TYPE ST_IPCDiagParamSpec :
STRUCT
	eParam: E_IPCDiag_ParameterKey;
	pData: PVOID;
	nSize: UDINT;
END_STRUCT
END_TYPE

(* stored: Version 1.1.0.1
   DUT ST_IPCDiagParamSpec: Id {9dbf62d2-8c08-037b-139c-5d4fff36e635} *)
